{attribute 'GeneratedUsingTerminal: EL1259-0000-0016'}
{attribute addProperty BoxType "EL1259-0000-0016"}
{attribute addProperty Id "StatusAT %I*Status_642C2ED16"}
{attribute addProperty CRC "1405132427"}
{attribute addProperty Size "6"}
TYPE MTO_Inputs_Channel_53C09E8B EXTENDS InputBase_8311D824 :
STRUCT
	{attribute addProperty Name "Status"}
	Status AT %I* : Status_642C2ED1;
END_STRUCT
END_TYPE

(* stored: Version 1.2.0.0, ProductVersion 3.1.4024.9
   DUT MTO_Inputs_Channel_53C09E8B: Id {f4b313c8-c7e9-4888-b4b9-65c3928d9c03} *)
